PROGRAM pouS1Prompts
VAR
END_VAR

// NETWORK 1

END_PROGRAM

(* stored: Version 1.1.0.1, ProductVersion 3.1.4024.12
   POU pouS1Prompts: Id {d0bcea03-d9bc-4b96-baec-8989514f2c5f}, SpecialFunc None *)
